# B&R Automation Studio project Splicer_V12_ACP10 (part 2)

#### slaveCyclic.st - Cyclic code
```iecst
(********************************************************************
 * COPYRIGHT -- Bernecker + Rainer
 ********************************************************************
 * Program: Slave_00
 * File: slaveCyclic.st
 * Author: Bernecker + Rainer
 * Created: March 01, 2011
 ********************************************************************
 * Implementation of program Slave_00
 ********************************************************************)

PROGRAM _CYCLIC

(************CHECK IF POWER SHOULD BE OFF ***************************)
    IF ((GlobalCommand.Power = FALSE) AND (Slave[SLAVE_INDEX].Command.Power = FALSE)) THEN
        SlaveStep := STATE_WAIT;
    END_IF

    (* central monitoring of the stop command allows a shorter reaction time *)
    IF ((GlobalCommand.Stop = TRUE) OR (Slave[SLAVE_INDEX].Command.Stop = TRUE)) THEN
        IF ((GlobalCommand.Power = TRUE) OR (Slave[SLAVE_INDEX].Command.Power = TRUE)) THEN
            SlaveStep := STATE_STOP;
            (* reset all FB execute inputs we use *)
            MC_Home_0.Execute := FALSE;
            MC_Halt_0.Execute := FALSE;
            MC_MoveAbsolute_0.Execute := FALSE;
            MC_MoveAdditive_0.Execute := FALSE;
            MC_MoveVelocity_0.Execute := FALSE;

            MC_BR_InitAutData_0.Execute := FALSE;
            MC_BR_AutCommand_0.Enable := FALSE;
            MC_BR_AutCommand_0.Start := FALSE;
            MC_BR_AutCommand_0.Restart := FALSE;
            MC_BR_AutCommand_0.Stop := FALSE;
            MC_BR_AutCommand_0.EndAutomat := FALSE;

            Slave[SLAVE_INDEX].Command.MoveJogPos := FALSE;
            Slave[SLAVE_INDEX].Command.MoveJogNeg := FALSE;
        END_IF
    END_IF

(************************** MC_READSTATUS ***************************)
MC_ReadStatus_0.Enable := NOT(MC_ReadStatus_0.Error);
MC_ReadStatus_0.Axis := SlaveRef[SLAVE_INDEX];
MC_ReadStatus_0();
Slave[SLAVE_INDEX].AxisState.Disabled             := MC_ReadStatus_0.Disabled;
Slave[SLAVE_INDEX].AxisState.StandStill           := MC_ReadStatus_0.StandStill;
Slave[SLAVE_INDEX].AxisState.Stopping             := MC_ReadStatus_0.Stopping;
Slave[SLAVE_INDEX].AxisState.Homing               := MC_ReadStatus_0.Homing;
Slave[SLAVE_INDEX].AxisState.DiscreteMotion       := MC_ReadStatus_0.DiscreteMotion;
Slave[SLAVE_INDEX].AxisState.ContinuousMotion     := MC_ReadStatus_0.ContinuousMotion;
Slave[SLAVE_INDEX].AxisState.SynchronizedMotion   := MC_ReadStatus_0.SynchronizedMotion;
Slave[SLAVE_INDEX].AxisState.ErrorStop            := MC_ReadStatus_0.Errorstop;

(********************** MC_BR_READDRIVESTATUS ***********************)
MC_BR_ReadDriveStatus_0.Enable := NOT(MC_BR_ReadDriveStatus_0.Error);
MC_BR_ReadDriveStatus_0.Axis := SlaveRef[SLAVE_INDEX];
MC_BR_ReadDriveStatus_0.AdrDriveStatus := ADR(Slave[SLAVE_INDEX].Status.DriveStatus);
MC_BR_ReadDriveStatus_0();

(********************* MC_READACTUALPOSITION ************************)
MC_ReadActualPosition_0.Enable := NOT(MC_ReadActualPosition_0.Error);
MC_ReadActualPosition_0.Axis := SlaveRef[SLAVE_INDEX];
MC_ReadActualPosition_0();
IF(MC_ReadActualPosition_0.Valid = TRUE) THEN
    Slave[SLAVE_INDEX].Status.ActPosition := MC_ReadActualPosition_0.Position;
END_IF

(********************* MC_READACTUALVELOCITY ************************)
MC_ReadActualVelocity_0.Enable := NOT(MC_ReadActualVelocity_0.Error);
MC_ReadActualVelocity_0.Axis := SlaveRef[SLAVE_INDEX];
MC_ReadActualVelocity_0();
IF(MC_ReadActualVelocity_0.Valid = TRUE) THEN
    Slave[SLAVE_INDEX].Status.ActVelocity := MC_ReadActualVelocity_0.Velocity;
END_IF

CASE SlaveStep OF
(****************************** WAIT ********************************)
    STATE_WAIT: (* STATE: Wait *)
        IF ((GlobalCommand.Power = TRUE) OR (Slave[SLAVE_INDEX].Command.Power = TRUE)) THEN
            SlaveStep := STATE_POWER_ON;
        ELSE
            MC_Power_0.Enable := FALSE;
        END_IF

        (* reset all FB execute inputs we use *)
        MC_Home_0.Execute := FALSE;
        MC_Halt_0.Execute := FALSE;
        MC_Stop_0.Execute := FALSE;
        MC_MoveAbsolute_0.Execute := FALSE;
        MC_MoveAdditive_0.Execute := FALSE;
        MC_MoveVelocity_0.Execute := FALSE;

        (* reset user commands *)
        Slave[SLAVE_INDEX].Command.Stop := FALSE;
        Slave[SLAVE_INDEX].Command.MoveJogPos := FALSE;
        Slave[SLAVE_INDEX].Command.MoveJogNeg := FALSE;
        Slave[SLAVE_INDEX].Command.MoveVelocity := FALSE;
        Slave[SLAVE_INDEX].Command.MoveAbsolute := FALSE;
        Slave[SLAVE_INDEX].Command.MoveAdditive := FALSE;

    (* End of STATE_WAIT *)

(****************************** POWER ON ****************************)
    STATE_POWER_ON: (* STATE: Power on *)
        IF (PowerSupplyOn = TRUE) THEN
            MC_Power_0.Enable := TRUE;
        END_IF
        IF (MC_Power_0.Status = TRUE) THEN
            SlaveStep := STATE_READY;
        END_IF

        (* if a power error occured switch off controller *)
        IF (MC_Power_0.Error = TRUE) THEN
            MC_Power_0.Enable := FALSE;
        END_IF

        (* End of STATE_POWER_ON *)

(****************************** READY *******************************)
    STATE_READY: (* STATE: Waiting for Commands *)
        IF ((Slave[SLAVE_INDEX].Command.Home = TRUE) OR (GlobalCommand.Home = TRUE)) THEN
            Slave[SLAVE_INDEX].Command.Home := FALSE;
            SlaveStep := STATE_HOME;
        ELSIF ((Slave[SLAVE_INDEX].Command.Stop = TRUE) OR (GlobalCommand.Stop = TRUE)) THEN
            SlaveStep := STATE_STOP;
        ELSIF (Slave[SLAVE_INDEX].Command.MoveJogPos = TRUE) THEN
            SlaveStep := STATE_JOG_POSITIVE;
        ELSIF (Slave[SLAVE_INDEX].Command.MoveJogNeg = TRUE) THEN
            SlaveStep := STATE_JOG_NEGATIVE;
        ELSIF (Slave[SLAVE_INDEX].Command.MoveAbsolute = TRUE) THEN
            Slave[SLAVE_INDEX].Command.MoveAbsolute := FALSE;
            SlaveStep := STATE_MOVE_ABSOLUTE;
        ELSIF (Slave[SLAVE_INDEX].Command.MoveAdditive = TRUE) THEN
            Slave[SLAVE_INDEX].Command.MoveAdditive := FALSE;
            SlaveStep := STATE_MOVE_ADDITIVE;
        ELSIF (Slave[SLAVE_INDEX].Command.MoveVelocity = TRUE) THEN
            Slave[SLAVE_INDEX].Command.MoveVelocity := FALSE;
            SlaveStep := STATE_MOVE_VELOCITY;
        ELSIF (Slave[SLAVE_INDEX].Command.Halt = TRUE) THEN
            Slave[SLAVE_INDEX].Command.Halt := FALSE;
            SlaveStep := STATE_HALT;
        ELSIF (Slave[SLAVE_INDEX].Command.StartAutomat = TRUE) THEN
            Slave[SLAVE_INDEX].Command.StartAutomat := FALSE;
            SlaveStep := STATE_AUTOMAT_INIT;
        ELSIF (Slave[SLAVE_INDEX].Command.RestartAutomat = TRUE) THEN
            Slave[SLAVE_INDEX].Command.RestartAutomat := FALSE;
            SlaveStep := STATE_AUTOMAT_RESTART;
        ELSIF (Slave[SLAVE_INDEX].Command.EndAutomat = TRUE) THEN
            Slave[SLAVE_INDEX].Command.EndAutomat := FALSE;
            SlaveStep := STATE_AUTOMAT_END;
        ELSIF (Slave[SLAVE_INDEX].Command.StopSlave = TRUE) THEN
            Slave[SLAVE_INDEX].Command.StopSlave := FALSE;
            SlaveStep := STATE_AUTOMAT_STOP;
        END_IF

        (* End of STATE_READY *)

(****************************** HOME ********************************)
    STATE_HOME: (* STATE: start homing process *)
        MC_Home_0.Position := Slave[SLAVE_INDEX].Parameter.HomePosition;
        MC_Home_0.HomingMode := Slave[SLAVE_INDEX].Parameter.HomeMode;
        MC_Home_0.Execute := TRUE;
        IF (MC_Home_0.Done = TRUE) THEN
            GlobalCommand.Home := FALSE;
            MC_Home_0.Execute := FALSE;
            SlaveStep := STATE_READY;
        END_IF

        (* if a homing error occured go to ready state *)
        IF ((MC_Home_0.Error = TRUE) OR (MC_Home_0.CommandAborted = TRUE)) THEN
            MC_Home_0.Execute := FALSE;
            SlaveStep := STATE_READY;
        END_IF

        (* End of STATE_HOME *)

(*************************** HALT MOVEMENT **************************)
    STATE_HALT: (* STATE: Stop the active movement *)
        MC_Halt_0.Deceleration := Slave[SLAVE_INDEX].Parameter.Deceleration;
        MC_Halt_0.Execute := TRUE;
        IF (MC_Halt_0.Done = TRUE) THEN
            MC_Halt_0.Execute := FALSE;
            SlaveStep := STATE_READY;
       END_IF

       (* check if error occured *)
       IF ((MC_Halt_0.Error = TRUE) OR (MC_Halt_0.CommandAborted = TRUE)) THEN
           MC_Halt_0.Execute := FALSE;
           SlaveStep := STATE_READY;
       END_IF

       (* End of STATE_HALT *)

(*************************** STOP MOVEMENT **************************)
    STATE_STOP: (* STATE: Stop movement as long as command is set *)
        MC_Stop_0.Deceleration := Slave[SLAVE_INDEX].Parameter.Deceleration;
        MC_Stop_0.Execute := TRUE;

        (* if axis is stopped go to ready state *)
        IF ((MC_Stop_0.Done = TRUE) AND (Slave[SLAVE_INDEX].Command.Stop = FALSE) AND (GlobalCommand.Stop = FALSE)) THEN
            MC_Stop_0.Execute := FALSE;
            SlaveStep := STATE_READY;
        END_IF

        (* check if error occured *)
        IF (((MC_Stop_0.Error = TRUE) OR (MC_Stop_0.CommandAborted = TRUE)) AND
             (Slave[SLAVE_INDEX].Command.Stop = FALSE) AND
             (GlobalCommand.Stop = FALSE)) THEN
            MC_Stop_0.Execute := FALSE;
            SlaveStep := STATE_READY;
        END_IF

       (* End of STATE_STOP *)

(******************* START JOG MOVEMENT POSITIVE ********************)
    STATE_JOG_POSITIVE: (* STATE: Start jog movement in positive direction *)
        MC_MoveVelocity_0.Velocity      := Slave[SLAVE_INDEX].Parameter.JogVelocity;
        MC_MoveVelocity_0.Acceleration  := Slave[SLAVE_INDEX].Parameter.Acceleration;
        MC_MoveVelocity_0.Deceleration  := Slave[SLAVE_INDEX].Parameter.Deceleration;
        MC_MoveVelocity_0.Direction     := mcPOSITIVE_DIR;
        MC_MoveVelocity_0.Execute := 1;

        (* check if jog movement should be stopped *)
        IF (Slave[SLAVE_INDEX].Command.MoveJogPos = FALSE) THEN
            MC_MoveVelocity_0.Execute := FALSE;
            SlaveStep := STATE_HALT;
        END_IF

        IF ((MC_MoveVelocity_0.Error = TRUE) OR (MC_MoveVelocity_0.CommandAborted = TRUE)) THEN
            MC_MoveVelocity_0.Execute := FALSE;
            SlaveStep := STATE_READY;
        END_IF

        (* End of STATE_JOG_POSITIVE *)

(********************START JOG MOVEMENT NEGATIVE ********************)
    STATE_JOG_NEGATIVE: (* STATE: Start jog movement in negative direction *)
        MC_MoveVelocity_0.Velocity      := Slave[SLAVE_INDEX].Parameter.JogVelocity;
        MC_MoveVelocity_0.Acceleration  := Slave[SLAVE_INDEX].Parameter.Acceleration;
        MC_MoveVelocity_0.Deceleration  := Slave[SLAVE_INDEX].Parameter.Deceleration;
        MC_MoveVelocity_0.Direction     := mcNEGATIVE_DIR;
        MC_MoveVelocity_0.Execute := 1;

        (* check if jog movement should be stopped *)
        IF (Slave[SLAVE_INDEX].Command.MoveJogNeg = FALSE) THEN
            MC_MoveVelocity_0.Execute := FALSE;
            SlaveStep := STATE_HALT;
        END_IF

        IF ((MC_MoveVelocity_0.Error = TRUE) OR (MC_MoveVelocity_0.CommandAborted = TRUE)) THEN
            MC_MoveVelocity_0.Execute := FALSE;
            SlaveStep := STATE_READY;
        END_IF

        (* End of STATE_JOG_NEGATIVE *)

(********************* START ABSOLUTE MOVEMENT **********************)
    STATE_MOVE_ABSOLUTE: (* STATE: Start absolute movement *)
        MC_MoveAbsolute_0.Position      := Slave[SLAVE_INDEX].Parameter.Position;
        MC_MoveAbsolute_0.Velocity      := Slave[SLAVE_INDEX].Parameter.Velocity;
        MC_MoveAbsolute_0.Acceleration  := Slave[SLAVE_INDEX].Parameter.Acceleration;
        MC_MoveAbsolute_0.Deceleration  := Slave[SLAVE_INDEX].Parameter.Deceleration;
        MC_MoveAbsolute_0.Direction     := Slave[SLAVE_INDEX].Parameter.Direction;
        MC_MoveAbsolute_0.Execute := 1;

        IF (Slave[SLAVE_INDEX].Command.Halt = TRUE) THEN
            Slave[SLAVE_INDEX].Command.Halt := 0;
            MC_MoveAbsolute_0.Execute := 0;
            SlaveStep := STATE_HALT;
        ELSIF (MC_MoveAbsolute_0.Done = TRUE) THEN
            MC_MoveAbsolute_0.Execute := FALSE;
            SlaveStep := STATE_READY;
        END_IF

        IF ((MC_MoveAbsolute_0.Error = TRUE) OR (MC_MoveAbsolute_0.CommandAborted = TRUE)) THEN
            MC_MoveAbsolute_0.Execute := FALSE;
            SlaveStep := STATE_READY;
        END_IF

        (* End of STATE_MOVE_ABSOLUTE *)

(********************* START ADDITIVE MOVEMENT **********************)
    STATE_MOVE_ADDITIVE: (* STATE: Start additive movement *)
        MC_MoveAdditive_0.Distance      := Slave[SLAVE_INDEX].Parameter.Distance;
        MC_MoveAdditive_0.Velocity      := Slave[SLAVE_INDEX].Parameter.Velocity;
        MC_MoveAdditive_0.Acceleration  := Slave[SLAVE_INDEX].Parameter.Acceleration;
        MC_MoveAdditive_0.Deceleration  := Slave[SLAVE_INDEX].Parameter.Deceleration;
        MC_MoveAdditive_0.Execute := 1;
        IF (Slave[SLAVE_INDEX].Command.Halt = TRUE) THEN
            Slave[SLAVE_INDEX].Command.Halt := FALSE;
            MC_MoveAdditive_0.Execute := FALSE;
            SlaveStep := STATE_HALT;
        ELSIF (MC_MoveAdditive_0.Done = TRUE) THEN
            MC_MoveAdditive_0.Execute := FALSE;
             SlaveStep := STATE_READY;
        END_IF

        (* check IF error occured *)
        IF ((MC_MoveAdditive_0.Error = TRUE) OR (MC_MoveAdditive_0.CommandAborted = TRUE)) THEN
            MC_MoveAdditive_0.Execute := FALSE;
            SlaveStep := STATE_READY;
        END_IF

        (* End of STATE_MOVE_ADDITIVE *)

(********************* START VELOCITY MOVEMENT **********************)
    STATE_MOVE_VELOCITY: (* STATE: Start velocity movement *)
        MC_MoveVelocity_0.Velocity      := Slave[SLAVE_INDEX].Parameter.Velocity;
        MC_MoveVelocity_0.Acceleration  := Slave[SLAVE_INDEX].Parameter.Acceleration;
        MC_MoveVelocity_0.Deceleration  := Slave[SLAVE_INDEX].Parameter.Deceleration;
        MC_MoveVelocity_0.Direction     := Slave[SLAVE_INDEX].Parameter.Direction;
        MC_MoveVelocity_0.Execute := 1;

        IF (Slave[SLAVE_INDEX].Command.Halt = TRUE) THEN
            Slave[SLAVE_INDEX].Command.Halt := FALSE;
            MC_MoveVelocity_0.Execute := FALSE;
            SlaveStep := STATE_HALT;
        ELSIF (MC_MoveVelocity_0.InVelocity = TRUE) THEN
            MC_MoveVelocity_0.Execute := FALSE;
             SlaveStep := STATE_READY;
        END_IF
        (* check if error occured *)
        IF ((MC_MoveVelocity_0.Error = TRUE) OR (MC_MoveVelocity_0.CommandAborted = TRUE)) THEN
            MC_MoveVelocity_0.Execute := FALSE;
            SlaveStep := STATE_READY;
        END_IF

        (* End of STATE_MOVE_ADDITIVE *)

(****************** INITIALIZE AUTOMAT PARAMETERS *******************)
    STATE_AUTOMAT_INIT:
        Labeler(MasterRef[0],AutData); (*Call of the function with the Automat Data*)

        MC_BR_InitAutData_0.InitOptions.GlobalParams      := mcALL_PARAMS;
        MC_BR_InitAutData_0.InitOptions.StateIndex        := mcALL_STATES;
        MC_BR_InitAutData_0.InitOptions.EventIndex        := mcALL_EVENTS;
        MC_BR_InitAutData_0.InitOptions.MaxStatesPerCycle := 14;
        MC_BR_InitAutData_0.InitOptions.Force             := mcOFF;
        MC_BR_InitAutData_0.AdrAutData  := ADR(AutData);
        MC_BR_InitAutData_0.Execute     := TRUE;

        (* wait for initialization done *)
        IF (MC_BR_InitAutData_0.Done = TRUE) THEN
            MC_BR_InitAutData_0.Execute := FALSE;
            SlaveStep := STATE_AUTOMAT_START;
        END_IF

        (* check if error occured *)
        IF (MC_BR_InitAutData_0.Error = TRUE) THEN
            MC_BR_InitAutData_0.Execute := FALSE;
            SlaveStep := STATE_READY;
        END_IF

        (* End of STATE_MOVE_VELOCITY *)

(********************** ENABLE CAM-AUTOMAT **************************)
    STATE_AUTOMAT_START:
        MC_BR_AutCommand_0.Enable := TRUE;
        MC_BR_AutCommand_0.Start := TRUE;

        (* wait for autoamt stop *)
        IF (Slave[SLAVE_INDEX].Command.Halt = TRUE) THEN
            Slave[SLAVE_INDEX].Command.Halt := FALSE;
            MC_BR_AutCommand_0.Enable := FALSE;
            MC_BR_AutCommand_0.Start := FALSE;
            SlaveStep := STATE_HALT;
        ELSIF (MC_BR_AutCommand_0.Running = TRUE) THEN
            MC_BR_AutCommand_0.Start := FALSE;
            SlaveStep := STATE_READY;
        END_IF

        (* check if error occured *)
        IF (MC_BR_AutCommand_0.Error = TRUE) THEN
            MC_BR_AutCommand_0.Enable := FALSE;
            MC_BR_AutCommand_0.Start := FALSE;
            SlaveStep := STATE_READY;
        END_IF

        (* End of STATE_AUTOMAT_START *)

(********************** RESTART CAM-AUTOMAT *************************)
    STATE_AUTOMAT_RESTART:
        IF (MC_BR_AutCommand_0.StandBy = FALSE) THEN
            SlaveStep := STATE_READY;
            RETURN;
        END_IF

        MC_BR_AutCommand_0.Enable := TRUE;
        MC_BR_AutCommand_0.Restart := TRUE;

        (* wait for autoamt stop *)
        IF (Slave[SLAVE_INDEX].Command.Halt = TRUE) THEN
            Slave[SLAVE_INDEX].Command.Halt := FALSE;
            MC_BR_AutCommand_0.Enable := FALSE;
            MC_BR_AutCommand_0.Restart := FALSE;
            SlaveStep := STATE_HALT;
        ELSIF (MC_BR_AutCommand_0.Running = TRUE) THEN
            MC_BR_AutCommand_0.Restart := FALSE;
            SlaveStep := STATE_READY;
        END_IF

        (* check if error occured *)
        IF (MC_BR_AutCommand_0.Error = TRUE) THEN
            MC_BR_AutCommand_0.Enable := FALSE;
            MC_BR_AutCommand_0.Restart := FALSE;
            SlaveStep := STATE_READY;
        END_IF

        (* End of STATE_AUTOMAT_RESTART *)

(*********************** STOP CAM-AUTOMAT ***************************)
    STATE_AUTOMAT_STOP:
        MC_BR_AutCommand_0.Deceleration := Slave[SLAVE_INDEX].Parameter.Deceleration;
        MC_BR_AutCommand_0.Stop := TRUE;

        (* check if automat is stopped *)
        IF (MC_BR_AutCommand_0.Running = FALSE) THEN
            MC_BR_AutCommand_0.Stop := FALSE;
            SlaveStep := STATE_READY;
        END_IF

        IF (MC_BR_AutCommand_0.Error = TRUE) THEN
            MC_BR_AutCommand_0.Enable := FALSE;
            MC_BR_AutCommand_0.Stop := FALSE;
            SlaveStep := STATE_READY;
        END_IF

        (* End of STATE_AUTOMAT_STOP *)

(************************ END CAM-AUTOMAT ***************************)
    STATE_AUTOMAT_END:
        MC_BR_AutCommand_0.Deceleration := Slave[SLAVE_INDEX].Parameter.Deceleration;
        MC_BR_AutCommand_0.Stop := TRUE;

        (* check if automat is stopped *)
        IF (MC_BR_AutCommand_0.Running = FALSE) THEN
            MC_BR_AutCommand_0.Enable := FALSE;
            MC_BR_AutCommand_0.EndAutomat := FALSE;
            SlaveStep := STATE_READY;
        END_IF

        (* check if error occured *)
        IF (MC_BR_AutCommand_0.Error = TRUE) THEN
            MC_BR_AutCommand_0.Enable := FALSE;
            MC_BR_AutCommand_0.EndAutomat := FALSE;
            SlaveStep := STATE_READY;
        END_IF

        (* End of STATE_AUTOMAT_STOP *)

(*********************** SEQUENCE END *******************************)
END_CASE

(*********************************************************************
        Function Block Calls
*********************************************************************)

(*************************** MC_POWER *******************************)
MC_Power_0.Axis := SlaveRef[SLAVE_INDEX];
MC_Power_0();

(**************************** MC_HOME *******************************)
MC_Home_0.Axis := SlaveRef[SLAVE_INDEX];
MC_Home_0();

(************************ MC_MOVEABSOLUTE ***************************)
MC_MoveAbsolute_0.Axis := SlaveRef[SLAVE_INDEX];
MC_MoveAbsolute_0();

(************************ MC_MOVEADDITIVE ***************************)
MC_MoveAdditive_0.Axis := SlaveRef[SLAVE_INDEX];
MC_MoveAdditive_0();

(************************ MC_MOVEVELOCITY ***************************)
MC_MoveVelocity_0.Axis := SlaveRef[SLAVE_INDEX];
MC_MoveVelocity_0();

(**************************** MC_STOP *******************************)
MC_Stop_0.Axis := SlaveRef[SLAVE_INDEX];
MC_Stop_0();

(*************************** MC_HALT ********************************)
MC_Halt_0.Axis := SlaveRef[SLAVE_INDEX];
MC_Halt_0();

(********************** MC_BR_INITAUTDATA ***************************)
MC_BR_InitAutData_0.Slave := SlaveRef[SLAVE_INDEX];
MC_BR_InitAutData_0();

(*********************** MC_BR_AUTCOMMAND ***************************)
MC_BR_AutCommand_0.SetSignal1 := Slave[SLAVE_INDEX].Command.SetSignal1;
MC_BR_AutCommand_0.SetSignal2 := Slave[SLAVE_INDEX].Command.SetSignal2;
MC_BR_AutCommand_0.SetSignal3 := Slave[SLAVE_INDEX].Command.SetSignal3;
MC_BR_AutCommand_0.SetSignal4 := Slave[SLAVE_INDEX].Command.SetSignal4;
MC_BR_AutCommand_0.ResetSignal1 := Slave[SLAVE_INDEX].Command.ResetSignal1;
MC_BR_AutCommand_0.ResetSignal2 := Slave[SLAVE_INDEX].Command.ResetSignal2;
MC_BR_AutCommand_0.ResetSignal3 := Slave[SLAVE_INDEX].Command.ResetSignal3;
MC_BR_AutCommand_0.ResetSignal4 := Slave[SLAVE_INDEX].Command.ResetSignal4;
MC_BR_AutCommand_0.Slave := SlaveRef[SLAVE_INDEX];
MC_BR_AutCommand_0();
Slave[SLAVE_INDEX].Status.AutomatRunning := MC_BR_AutCommand_0.Running;
Slave[SLAVE_INDEX].Status.AutomatStandBy := MC_BR_AutCommand_0.StandBy;
Slave[SLAVE_INDEX].Status.ActualStateIndex := MC_BR_AutCommand_0.ActualStateIndex;
Slave[SLAVE_INDEX].Status.ActualStateCamIndex := MC_BR_AutCommand_0.ActualStateCamIndex;
Slave[SLAVE_INDEX].Status.InCam := MC_BR_AutCommand_0.InCam;
Slave[SLAVE_INDEX].Status.InCompensation := MC_BR_AutCommand_0.InCompensation;
END_PROGRAM
```

#### slaveInit.st - Initialization code
```iecst
(********************************************************************
 * COPYRIGHT -- Bernecker + Rainer
 ********************************************************************
 * Program: Slave_00
 * File: slaveInit.st
 * Author: Bernecker + Rainer
 * Created: March 01, 2011
 ********************************************************************
 * Implementation of program Slave_00
 ********************************************************************)

PROGRAM _INIT
SlaveStep := STATE_WAIT; (* start step *)

Slave[SLAVE_INDEX].Parameter.Velocity       := 1000; (* velocity for movement *)
Slave[SLAVE_INDEX].Parameter.Acceleration   := 5000; (* acceleration for movement *)
Slave[SLAVE_INDEX].Parameter.Deceleration   := 5000; (* deceleration for movement *)
Slave[SLAVE_INDEX].Parameter.JogVelocity    := 400;  (* velocity for jogging *)
END_PROGRAM
```

#### slave.var - Local variables
```iecst
(*Actual step inside step sequencer*)
VAR
	SlaveStep : USINT; (*current  step in the step sequence*)
END_VAR
VAR CONSTANT
	STATE_WAIT : USINT := 0; (*constant for a waiting step*)
	STATE_POWER_ON : USINT := 1; (*constant for the step in which the controller is switched on*)
	STATE_HOME : USINT := 2; (*constant for the step in which the axis is referenced*)
	STATE_READY : USINT := 10; (*constant for a waiting step*)
	STATE_HALT : USINT := 11; (*constant for the step in which movements are stopped*)
	STATE_STOP : USINT := 12; (*constant for the step in which movements are stopped*)
	STATE_JOG_POSITIVE : USINT := 13; (*constant for the step in which positive jogging movement is executed*)
	STATE_JOG_NEGATIVE : USINT := 14; (*constant for the step in which negative jogging movement is executed*)
	STATE_MOVE_ABSOLUTE : USINT := 15; (*constant for the step in which a movement to defined position is executed*)
	STATE_MOVE_ADDITIVE : USINT := 16; (*constant for the step in which a movement with defined distance is executed*)
	STATE_MOVE_VELOCITY : USINT := 17; (*constant for the step in which a movement with defined velocity is started*)
	STATE_AUTOMAT_INIT : USINT := 30; (*constant for the step in which the automat is configured*)
	STATE_AUTOMAT_START : USINT := 31; (*constant for the step in which the automat is started*)
	STATE_AUTOMAT_STOP : USINT := 32; (*constant for the step in which the automat is stopped*)
	STATE_AUTOMAT_RESTART : USINT := 33; (*constant for the step in which the automat is restarted*)
	STATE_AUTOMAT_END : USINT := 34; (*constant for the step in which the automat is finished*)
END_VAR
(*Index of the used axis*)
VAR CONSTANT
	SLAVE_INDEX : USINT := 0; (*Index of the used axis*)
END_VAR
(*Configuration data of the automat*)
VAR
	AutData : MC_AUTDATA_TYP; (*configuration of the automat*)
END_VAR
(*Function Blocks*)
VAR
	MC_BR_AutCommand_0 : MC_BR_AutCommand; (*Function Block*)
	MC_BR_InitAutData_0 : MC_BR_InitAutData; (*Function Block*)
	MC_BR_ReadDriveStatus_0 : MC_BR_ReadDriveStatus; (*Function Block *)
	MC_Halt_0 : MC_Halt; (*Function Block *)
	MC_Home_0 : MC_Home; (*Function Block *)
	MC_MoveAbsolute_0 : MC_MoveAbsolute; (*Function Block *)
	MC_MoveAdditive_0 : MC_MoveAdditive; (*Function Block *)
	MC_MoveVelocity_0 : MC_MoveVelocity; (*Function Block *)
	MC_Power_0 : MC_Power; (*Function Block *)
	MC_ReadActualPosition_0 : MC_ReadActualPosition; (*Function Block *)
	MC_ReadActualVelocity_0 : MC_ReadActualVelocity; (*Function Block *)
	MC_ReadStatus_0 : MC_ReadStatus; (*Function Block *)
	MC_Stop_0 : MC_Stop; (*Function Block *)
END_VAR
```

#### slave.fun - functions
```iecst
(********************************************************************
 * COPYRIGHT -- Bernecker + Rainer
 ********************************************************************
 * Program: Slave_00
 * File: Slave_00.fun
 * Author: reischlj
 * Created: March 09, 2011
 ********************************************************************
 * Functions and function blocks of program Slave_00
 ********************************************************************)

FUNCTION Labeler : BOOL
	VAR_INPUT
		Axis : UDINT;
	END_VAR
	VAR_IN_OUT
		AutData : MC_AUTDATA_TYP;
	END_VAR
END_FUNCTION

FUNCTION CrossCutter : BOOL
	VAR_INPUT
		Axis : UDINT;
	END_VAR
	VAR_IN_OUT
		AutData : MC_AUTDATA_TYP;
	END_VAR
END_FUNCTION

FUNCTION FlyingSaw : BOOL
	VAR_INPUT
		Axis  : UDINT;
	END_VAR
	VAR_IN_OUT
		AutData : MC_AUTDATA_TYP;
	END_VAR
END_FUNCTION
```

#### Labeler.st - function
```iecst
(********************************************************************
 * COPYRIGHT -- Bernecker + Rainer
 ********************************************************************
 * PROGRAM: Slave
 * File: Labeler.st
 * Author: Bernecker + Rainer
 * Created: March 01, 2011
 *******************************************************************)

FUNCTION Labeler
    (*general automat parameter*)
        AutData.Master              := Axis;

        AutData.MaxMasterVelocity   := 1000;

    (*Automat STATE 0 Basis State*)

        AutData.State[0].Event[0].Type      := ncST_END;

        AutData.State[0].Event[0].Attribute := ncAT_ONCE;

        AutData.State[0].Event[0].NextState := 1;

    (*Automat STATE 1 Standstill*)

        AutData.State[1].CamProfileIndex    := 16#FFFF;

        AutData.State[1].MasterFactor       := 200;

        AutData.State[1].SlaveFactor        := 0;

        AutData.State[1].CompMode           := ncONLYCOMP;

        AutData.State[1].MasterCompDistance := 800;

        AutData.State[1].SlaveCompDistance  := 0;

        AutData.State[1].Event[0].Type      := ncTRIGGER1+ncP_EDGE;

        AutData.State[1].Event[0].Attribute := ncST_END;

        AutData.State[1].Event[0].NextState := 2;

        AutData.State[1].Event[1].Type      := ncST_END;

        AutData.State[1].Event[1].Attribute := ncST_END;

        AutData.State[1].Event[1].NextState := 1;

    (*Automat STATE 2 Labeling with half compensation*)

        AutData.State[2].CamProfileIndex    := 16#FFFF;

        AutData.State[2].MasterFactor       := 200;

        AutData.State[2].SlaveFactor        := 200;

        AutData.State[2].CompMode           := ncONLYCOMP;
        AutData.State[2].MasterCompDistance := 800;

        AutData.State[2].SlaveCompDistance  := 400;

        AutData.State[2].Event[0].Type      := ncTRIGGER1+ncP_EDGE;

        AutData.State[2].Event[0].Attribute := ncST_END;

        AutData.State[2].Event[0].NextState := 3;

        AutData.State[2].Event[1].Type      := ncST_END;

        AutData.State[2].Event[1].Attribute := ncST_END;

        AutData.State[2].Event[1].NextState := 4;

    (*Automat STATE 3 Labeling *)

        AutData.State[3].CamProfileIndex    := 16#FFFF;

        AutData.State[3].MasterFactor       := 200;

        AutData.State[3].SlaveFactor        := 200;

        AutData.State[3].CompMode           := ncONLYCOMP;

        AutData.State[3].MasterCompDistance := 800;

        AutData.State[3].SlaveCompDistance  := 800;

        AutData.State[3].Event[0].Type      := ncTRIGGER1+ncP_EDGE;

        AutData.State[3].Event[0].Attribute := ncST_END;

        AutData.State[3].Event[0].NextState := 3;

        AutData.State[3].Event[1].Type      := ncST_END;
		AutData.State[3].Event[1].Attribute := ncST_END;
		AutData.State[3].Event[1].NextState := 4;

    (*Automat STATE 4 Return to starting position*)
        AutData.State[4].CamProfileIndex    := 16#FFFF;
        AutData.State[4].MasterFactor       := 200;
        AutData.State[4].SlaveFactor        := 0;
        AutData.State[4].CompMode           := ncONLYCOMP;
        AutData.State[4].MasterCompDistance := 800;
        AutData.State[4].SlaveCompDistance  := 400;

        AutData.State[4].Event[0].Type      := ncTRIGGER1+ncP_EDGE;
        AutData.State[4].Event[0].Attribute := ncST_END;
        AutData.State[4].Event[0].NextState := 2;

        AutData.State[4].Event[1].Type      := ncST_END;
        AutData.State[4].Event[1].Attribute := ncST_END;
        AutData.State[4].Event[1].NextState := 1;

        Labeler := TRUE;
END_FUNCTION
```

#### CrossCutter.st - function
```iecst
(********************************************************************
 * COPYRIGHT -- Bernecker + Rainer
 ********************************************************************
 * PROGRAM: Slave
 * File: CrossCutter.st
 * Author: Bernecker + Rainer
 * Created: March 01, 2011
 *******************************************************************)

FUNCTION CrossCutter
    (*general automat parameter*)
        AutData.Master              := Axis;

        AutData.MaxMasterVelocity   := 1000;

    (*Automat STATE 0 Basis State*)

        AutData.State[0].Event[0].Type      := ncST_END;

        AutData.State[0].Event[0].Attribute := ncAT_ONCE;

        AutData.State[0].Event[0].NextState := 1;

    (*Automat STATE 1 Standstill*)

        AutData.State[1].CamProfileIndex    := 16#FFFE;

        AutData.State[1].MasterFactor       := 200;

        AutData.State[1].SlaveFactor        := 0;
        AutData.State[1].CompMode           := ncWITH_CAM;
        AutData.State[1].MasterCompDistance := 1000;
        AutData.State[1].SlaveCompDistance  := 0;

        AutData.State[1].Event[0].Type      := ncSIGNAL1;
        AutData.State[1].Event[0].Attribute := ncAT_ONCE;
        AutData.State[1].Event[0].NextState := 2;

    (*Automat STATE 2 Move Slave to Cutting Position*)
        AutData.State[2].CamProfileIndex    := 16#FFFF;
        AutData.State[2].MasterFactor       := 200;
        AutData.State[2].SlaveFactor        := 200;
        AutData.State[2].CompMode           := ncWITH_CAM;
        AutData.State[2].MasterCompDistance := 500;
        AutData.State[2].SlaveCompDistance  := 1800;

        AutData.State[2].Event[0].Type      := ncST_END;
        AutData.State[2].Event[0].Attribute := ncST_END;
        AutData.State[2].Event[0].NextState := 3;

    (*Automat STATE 3 Execute one cut every master period*)
        AutData.State[3].CamProfileIndex    := 16#FFFF;
        AutData.State[3].MasterFactor       := 200;
        AutData.State[3].SlaveFactor        := 200;
        AutData.State[3].CompMode           := ncWITH_CAM;
        AutData.State[3].MasterCompDistance := 1000;
        AutData.State[3].SlaveCompDistance  := 3600;

        AutData.State[3].Event[0].Type      := ncSIGNAL2;
        AutData.State[3].Event[0].Attribute := ncST_END;
        AutData.State[3].Event[0].NextState := 4;

        AutData.State[3].Event[1].Type      := ncST_END;
        AutData.State[3].Event[1].Attribute := ncST_END;
        AutData.State[3].Event[1].NextState := 3;

    (*Automat STATE 4 Stop Motion at Starting Point*)
        AutData.State[4].CamProfileIndex    := 16#FFFF;
        AutData.State[4].MasterFactor       := 200;
        AutData.State[4].SlaveFactor        := 0;
        AutData.State[4].CompMode           := ncWITH_CAM;
        AutData.State[4].MasterCompDistance := 500;
        AutData.State[4].SlaveCompDistance  := 1800;

        AutData.State[4].Event[0].Type      := ncST_END;
        AutData.State[4].Event[0].Attribute := ncST_END;
        AutData.State[4].Event[0].NextState := 1;

        CrossCutter := TRUE;
END_FUNCTION
```

#### FlyingSaw.st - function
```iecst
(********************************************************************
 * COPYRIGHT -- Bernecker + Rainer
 ********************************************************************
 * PROGRAM: Slave
 * File: FlyingSaw.st
 * Author: Bernecker + Rainer
 * Created: March 01, 2011
 *******************************************************************)

FUNCTION FlyingSaw
    (*general automat parameters*)
        AutData.Master              := Axis;

        AutData.StartPosition       := 0;

        AutData.StartInterval       := 1000;

        AutData.MaxMasterVelocity   := 1000;

    (*Automat STATE 0 Basis State*)

        AutData.State[0].Event[0].Type      := ncST_END;

        AutData.State[0].Event[0].Attribute := ncAT_ONCE;

        AutData.State[0].Event[0].NextState := 1;

    (*Automat STATE 1 Standstill*)

        AutData.State[1].CamProfileIndex    := 16#FFFF;

        AutData.State[1].MasterFactor       := 200;

        AutData.State[1].SlaveFactor        := 0;

        AutData.State[1].CompMode           := ncONLYCOMP;

        AutData.State[1].MasterCompDistance := 800;

        AutData.State[1].SlaveCompDistance  := 0;

        AutData.State[1].Event[0].Type      := ncS_START;

        AutData.State[1].Event[0].Attribute := ncAT_ONCE;

        AutData.State[1].Event[0].NextState := 2;

    (*Autoamt STATE 2 Synchronous movement*)
        AutData.State[2].CamProfileIndex    := 16#FFFF;
        AutData.State[2].MasterFactor       := 500;
        AutData.State[2].SlaveFactor        := 500;
        AutData.State[2].CompMode           := ncONLYCOMP;
        AutData.State[2].MasterCompDistance := 100;
        AutData.State[2].SlaveCompDistance  := 100;

        AutData.State[2].Event[0].Type      := ncST_END;
        AutData.State[2].Event[0].Attribute := ncST_END;
        AutData.State[2].Event[0].NextState := 3;

    (*Automat STATE 3 Return to starting position*)
        AutData.State[3].CamProfileIndex    := 16#FFFF;
        AutData.State[3].MasterFactor       := 100;
        AutData.State[3].SlaveFactor        := 0;
        AutData.State[3].CompMode           := ncONLYCOMP;
        AutData.State[3].MasterCompDistance := 800;
        AutData.State[3].SlaveCompDistance  := -600;

        AutData.State[3].Event[0].Type      := ncST_END;
        AutData.State[3].Event[0].Attribute := ncST_END;
        AutData.State[3].Event[0].NextState := 1;

        FlyingSaw := TRUE;
END_FUNCTION
```

### Program Logical/Template/Logical/LibACP10MC_MotionControl_ST/ErrorHandling (IEC) - error handling task

#### errorHandlingCyclic.st - Cyclic code
```iecst
(********************************************************************
 * COPYRIGHT -- Bernecker + Rainer
 ********************************************************************
 * Program: ErrorHandling
 * File: errorHandlingCyclic.st
 * Author: Bernecker + Rainer
 * Created: March 01, 2011
 ********************************************************************
 * Implementation of program Errorhandling
 ********************************************************************)

PROGRAM _CYCLIC

(******************************ERROR_CHECK***************************)
(* check if one of the used FBs reports an error *)
IF ((MC_BR_AxisErrorCollector_0.Error = TRUE) OR (MC_Reset_0.Error = TRUE)) THEN
    ErrorStep := STATE_INTERNAL_ERROR;
END_IF

FOR configAxisIndex := 0 TO TOTAL_AXES BY 1 DO
    IF ((MC_BR_ReadAxisError_0[configAxisIndex].Error = TRUE) OR (MC_ReadStatus_0[configAxisIndex].Error = TRUE)) THEN
        ErrorStep := STATE_INTERNAL_ERROR;
        EXIT;
    END_IF
END_FOR

CASE ErrorStep OF

(**************************** CONFIGURATE_FBS ***********************)
    STATE_CONFIG_FBS: (* configurate the used FBs for the error handling *)
        MC_BR_AxisErrorCollector_0.Axis := mcALL_AXES;
        MC_BR_AxisErrorCollector_0.Enable := TRUE;

        (* configuration the MC_BR_ReadAxisError_0-FBs for all single axes *)
        FOR axisIndex := 0 TO (AXIS_MAX_INDEX) BY 1 DO
            MC_BR_ReadAxisError_0[axisIndex].Axis := AxisRef[axisIndex];
            MC_BR_ReadAxisError_0[axisIndex].Enable := TRUE;
            MC_BR_ReadAxisError_0[axisIndex].Configuration.Format := mcWRAP;
            MC_BR_ReadAxisError_0[axisIndex].Configuration.LineLength := SIZEOF(Axis[axisIndex].Error.ErrorText[0]);
            MC_BR_ReadAxisError_0[axisIndex].Configuration.DataLength := SIZEOF(Axis[axisIndex].Error.ErrorText);
            MC_BR_ReadAxisError_0[axisIndex].Configuration.DataAddress := ADR(Axis[axisIndex].Error.ErrorText[0]);
            MC_BR_ReadAxisError_0[axisIndex].Configuration.DataObjectName :='acp10etxen';
            MC_BR_ReadAxisError_0[axisIndex].Mode := mcTEXT;

            MC_ReadStatus_0[axisIndex].Axis := AxisRef[axisIndex];
            MC_ReadStatus_0[axisIndex].Enable := TRUE;
        END_FOR

        (* configuration the MC_BR_ReadAxisError_0-FBs for all master axes *)
        FOR masterIndex := 0 TO (MASTER_MAX_INDEX) BY 1 DO
            MC_BR_ReadAxisError_0[masterIndex+AXIS_NUMBER].Axis := MasterRef[masterIndex];
            MC_BR_ReadAxisError_0[masterIndex+AXIS_NUMBER].Enable := TRUE;
            MC_BR_ReadAxisError_0[masterIndex+AXIS_NUMBER].Configuration.Format := mcWRAP;
            MC_BR_ReadAxisError_0[masterIndex+AXIS_NUMBER].Configuration.LineLength := SIZEOF(Master[masterIndex].Error.ErrorText[0]);
            MC_BR_ReadAxisError_0[masterIndex+AXIS_NUMBER].Configuration.DataLength := SIZEOF(Master[masterIndex].Error.ErrorText);
            MC_BR_ReadAxisError_0[masterIndex+AXIS_NUMBER].Configuration.DataAddress := ADR(Master[masterIndex].Error.ErrorText[0]);
            MC_BR_ReadAxisError_0[masterIndex+AXIS_NUMBER].Configuration.DataObjectName := 'acp10etxen';
            MC_BR_ReadAxisError_0[masterIndex+AXIS_NUMBER].Mode := mcTEXT;

            MC_ReadStatus_0[masterIndex+AXIS_NUMBER].Axis := MasterRef[masterIndex];
            MC_ReadStatus_0[masterIndex+AXIS_NUMBER].Enable := TRUE;
        END_FOR

        (* configuration the MC_BR_ReadAxisError_0-FBs for all slave axes *)
        FOR slaveIndex := 0 TO (SLAVE_MAX_INDEX) BY 1 DO
            MC_BR_ReadAxisError_0[slaveIndex+AXIS_NUMBER+MASTER_NUMBER].Axis := SlaveRef[slaveIndex];
            MC_BR_ReadAxisError_0[slaveIndex+AXIS_NUMBER+MASTER_NUMBER].Enable := TRUE;
            MC_BR_ReadAxisError_0[slaveIndex+AXIS_NUMBER+MASTER_NUMBER].Configuration.Format := mcWRAP;
            MC_BR_ReadAxisError_0[slaveIndex+AXIS_NUMBER+MASTER_NUMBER].Configuration.LineLength := SIZEOF(Slave[slaveIndex].Error.ErrorText[0]);
            MC_BR_ReadAxisError_0[slaveIndex+AXIS_NUMBER+MASTER_NUMBER].Configuration.DataLength := SIZEOF(Slave[slaveIndex].Error.ErrorText);
            MC_BR_ReadAxisError_0[slaveIndex+AXIS_NUMBER+MASTER_NUMBER].Configuration.DataAddress := ADR(Slave[slaveIndex].Error.ErrorText[0]);
            MC_BR_ReadAxisError_0[slaveIndex+AXIS_NUMBER+MASTER_NUMBER].Configuration.DataObjectName := 'acp10etxen';
            MC_BR_ReadAxisError_0[slaveIndex+AXIS_NUMBER+MASTER_NUMBER].Mode := mcTEXT;

            MC_ReadStatus_0[slaveIndex+AXIS_NUMBER+MASTER_NUMBER].Axis := SlaveRef[slaveIndex];
            MC_ReadStatus_0[slaveIndex+AXIS_NUMBER+MASTER_NUMBER].Enable := TRUE;
        END_FOR

        (* configuration the MC_BR_ReadAxisError_0-FBs for all power supply module *)
        FOR psmIndex := 0 TO (PSM_MAX_INDEX) BY 1 DO
            MC_BR_ReadAxisError_0[psmIndex+AXIS_NUMBER+MASTER_NUMBER+SLAVE_NUMBER].Axis := PsmRef[psmIndex];
            MC_BR_ReadAxisError_0[psmIndex+AXIS_NUMBER+MASTER_NUMBER+SLAVE_NUMBER].Enable := TRUE;
            MC_BR_ReadAxisError_0[psmIndex+AXIS_NUMBER+MASTER_NUMBER+SLAVE_NUMBER].Configuration.Format := mcWRAP;
            MC_BR_ReadAxisError_0[psmIndex+AXIS_NUMBER+MASTER_NUMBER+SLAVE_NUMBER].Configuration.LineLength := SIZEOF(PowerSupply[psmIndex].Error.ErrorText[0]);
            MC_BR_ReadAxisError_0[psmIndex+AXIS_NUMBER+MASTER_NUMBER+SLAVE_NUMBER].Configuration.DataLength := SIZEOF(PowerSupply[psmIndex].Error.ErrorText);
            MC_BR_ReadAxisError_0[psmIndex+AXIS_NUMBER+MASTER_NUMBER+SLAVE_NUMBER].Configuration.DataAddress := ADR(PowerSupply[psmIndex].Error.ErrorText[0]);
            MC_BR_ReadAxisError_0[psmIndex+AXIS_NUMBER+MASTER_NUMBER+SLAVE_NUMBER].Configuration.DataObjectName := 'acp10etxen';
            MC_BR_ReadAxisError_0[psmIndex+AXIS_NUMBER+MASTER_NUMBER+SLAVE_NUMBER].Mode := mcTEXT;

            MC_ReadStatus_0[psmIndex+AXIS_NUMBER+MASTER_NUMBER+SLAVE_NUMBER].Axis := PsmRef[psmIndex];
            MC_ReadStatus_0[psmIndex+AXIS_NUMBER+MASTER_NUMBER+SLAVE_NUMBER].Enable := TRUE;
        END_FOR

        ErrorStep := STATE_WAIT;
        AcknowledgeStep := STATE_ERROR_SCAN;

        (* End of STATE_CONFIG_FBS *)

(*************************** CHECK_AXES_FOR_ERROR *******************)
    STATE_WAIT: (* check if at least on one of the axes an error occured *)
        IF ((MC_BR_AxisErrorCollector_0.AxisError = TRUE) OR
            (MC_BR_AxisErrorCollector_0.AxisWarning = TRUE) OR
            (MC_BR_AxisErrorCollector_0.FunctionBlockError = TRUE) OR
            (MC_BR_AxisErrorCollector_0.Errorstop = TRUE)) THEN
              ErrorStep := STATE_ERROR_HANDLING;
        ELSE
            GlobalError.AxisTyp := '';
            GlobalError.AxisIndex := 0;
            GlobalError.ErrorRecord.Info := 0;
            GlobalError.ErrorRecord.Number := 0;
            GlobalError.ErrorRecord.ParID := 0;
            GlobalError.ErrorText[0] := '';
            GlobalError.ErrorText[1] := '';
            GlobalError.ErrorText[2] := '';
            GlobalError.ErrorText[3] := '';
        END_IF

        (* End of STATE_WAIT *)

(**************************** HANDLE_ACTIVE_ERRORS ******************)
    STATE_ERROR_HANDLING: (* check witch axis is in ErrorStop and withc axes has to be stopped *)
        (* check if a single axis has to be stopped *)
        FOR axisIndex := 0 TO (AXIS_MAX_INDEX) BY 1 DO
            IF (MC_ReadStatus_0[axisIndex].Errorstop = TRUE) THEN
                Axis[axisIndex].Command.Stop := TRUE;
            END_IF
        END_FOR

        (* check if the master slave combination has to be stopped *)
        FOR masterIndex := 0 TO (MASTER_MAX_INDEX) BY 1 DO
            IF (MC_ReadStatus_0[masterIndex+AXIS_NUMBER].Errorstop = TRUE) THEN
                FOR masterIndex := 0 TO (MASTER_MAX_INDEX) BY 1 DO
                    Master[masterIndex].Command.Stop := TRUE;
                END_FOR

                FOR slaveIndex := 0 TO (SLAVE_MAX_INDEX) BY 1 DO
                    Slave[slaveIndex].Command.Stop := TRUE;
                END_FOR
            END_IF
        END_FOR

        (* check if the master slave combination has to be stopped *)
        FOR slaveIndex := 0 TO (SLAVE_MAX_INDEX) BY 1 DO
            IF  (MC_ReadStatus_0[slaveIndex+AXIS_NUMBER+MASTER_NUMBER].Errorstop = TRUE) THEN
                FOR masterIndex := 0 TO (MASTER_MAX_INDEX) BY 1 DO
                    Master[masterIndex].Command.Stop := TRUE;
                END_FOR

                FOR slaveIndex := 0 TO (SLAVE_MAX_INDEX) BY 1 DO
                    Slave[slaveIndex].Command.Stop := TRUE;
                END_FOR
            END_IF
        END_FOR

    (******************* STEP_SEQUENCE OF ERROR ACKNOWLEDGE *************)
    CASE AcknowledgeStep OF
        (************************** SEARCH FOR ERRORS ***********************)
        STATE_ERROR_SCAN: (* check if an error is active on one of the axis *)
            ErrorStep := STATE_WAIT;
            FOR totalAxisIndex := 0 TO (TOTAL_AXES-1) BY 1 DO
                IF ((MC_BR_ReadAxisError_0[totalAxisIndex].AxisErrorCount > 0) OR
                    (MC_BR_ReadAxisError_0[totalAxisIndex].AxisWarningCount > 0) OR
                    (MC_BR_ReadAxisError_0[totalAxisIndex].FunctionBlockErrorCount > 0)) THEN
                    AcknowledgeStep := STATE_ERROR_ACKNOWLEDGE;
                    ErrorStep := STATE_ERROR_HANDLING;
                    EXIT;
                ELSIF (MC_ReadStatus_0[totalAxisIndex].Errorstop = TRUE) THEN
                    AcknowledgeStep := STATE_RESET;
                    ErrorStep := STATE_ERROR_HANDLING;
                    EXIT;
                END_IF
            END_FOR

            (* End of STATE_ERROR_SCAN *)

        (********************** WAIT FOR ACKNOWLEDGE ************************)
        STATE_ERROR_ACKNOWLEDGE:
            (* copy the actual error information to the global error structure *)
            IF (totalAxisIndex < AXIS_NUMBER) THEN
                GlobalError.AxisTyp := 'Axis';
                GlobalError.ErrorText := Axis[totalAxisIndex].Error.ErrorText;
                GlobalError.ErrorRecord := Axis[totalAxisIndex].Error.ErrorRecord;
            ELSIF (totalAxisIndex < (AXIS_NUMBER+MASTER_NUMBER)) THEN
                GlobalError.AxisTyp := 'Master';
                GlobalError.ErrorText := Master[totalAxisIndex-AXIS_NUMBER].Error.ErrorText;
                GlobalError.ErrorRecord := Master[totalAxisIndex-AXIS_NUMBER].Error.ErrorRecord;
            ELSIF (totalAxisIndex < (AXIS_NUMBER+MASTER_NUMBER+SLAVE_NUMBER)) THEN
                GlobalError.AxisTyp := 'Slave';
                GlobalError.ErrorText := Slave[totalAxisIndex-(AXIS_NUMBER+MASTER_NUMBER)].Error.ErrorText;
                GlobalError.ErrorRecord := Slave[totalAxisIndex-(AXIS_NUMBER+MASTER_NUMBER)].Error.ErrorRecord;
            ELSIF (totalAxisIndex < (AXIS_NUMBER+MASTER_NUMBER+SLAVE_NUMBER+PSM_NUMBER)) THEN
                GlobalError.AxisTyp := 'PSM';
                GlobalError.ErrorText := PowerSupply[totalAxisIndex-(AXIS_NUMBER+MASTER_NUMBER+SLAVE_NUMBER)].Error.ErrorText;
                GlobalError.ErrorRecord := PowerSupply[totalAxisIndex-(AXIS_NUMBER+MASTER_NUMBER+SLAVE_NUMBER)].Error.ErrorRecord;
            END_IF
            GlobalError.AxisIndex := totalAxisIndex;

            IF (GlobalCommand.ErrorAcknowledge = TRUE) THEN
                GlobalCommand.ErrorAcknowledge := FALSE;
                MC_BR_ReadAxisError_0[totalAxisIndex].Acknowledge := TRUE;
            ELSIF (MC_BR_ReadAxisError_0[totalAxisIndex].Acknowledge = TRUE) THEN
                MC_BR_ReadAxisError_0[totalAxisIndex].Acknowledge := FALSE;
                AcknowledgeStep := STATE_ERROR_SCAN;
            END_IF

            (* End of STATE_ERROR_ACKNOWLEDGE *)

        (************************* RESET AXES IN ERRORSTEP ******************)
        STATE_RESET:
            IF (totalAxisIndex < AXIS_NUMBER) THEN
                MC_Reset_0.Axis := AxisRef[totalAxisIndex];
            ELSIF (totalAxisIndex < (AXIS_NUMBER+MASTER_NUMBER)) THEN
                MC_Reset_0.Axis := MasterRef[totalAxisIndex-AXIS_NUMBER];
            ELSIF (totalAxisIndex < (AXIS_NUMBER+MASTER_NUMBER+SLAVE_NUMBER)) THEN
                MC_Reset_0.Axis := SlaveRef[totalAxisIndex-(AXIS_NUMBER+MASTER_NUMBER)];
            ELSE
                MC_Reset_0.Axis := PsmRef[totalAxisIndex-(AXIS_NUMBER+MASTER_NUMBER+SLAVE_NUMBER)];
            END_IF
            MC_Reset_0.Execute := TRUE;

            IF (MC_Reset_0.Done = TRUE) THEN
                MC_Reset_0.Execute := 0;
                AcknowledgeStep := STATE_ERROR_SCAN;
            END_IF

            (* End of STATE_RESET *)
    END_CASE
    (************* END OF STEP SEQUENCE OF ERROR ACKNOWLEDGE ************)

    (* End of STATE_ERROR_HANDLING *)

(****************** DEACTIVATE USED FBS IN CASE OF ERROR ************)
    STATE_INTERNAL_ERROR:
        MC_BR_AxisErrorCollector_0.Enable := FALSE;
        MC_Reset_0.Execute := FALSE;

        FOR configAxisIndex := 0 TO (TOTAL_AXES-1) BY 1 DO
            MC_BR_ReadAxisError_0[configAxisIndex].Enable := FALSE;
            MC_ReadStatus_0[configAxisIndex].Enable := FALSE;
        END_FOR

        ErrorStep := STATE_CONFIG_FBS;

        (* End of STATE_INTERNAL_ERROR *)

END_CASE

(************************** CALL FBS ********************************)
MC_BR_AxisErrorCollector_0();

FOR configAxisIndex := 0 TO TOTAL_AXES BY 1 DO
    MC_BR_ReadAxisError_0[configAxisIndex]();
    IF (configAxisIndex < AXIS_NUMBER) THEN
        Axis[configAxisIndex].Error.AxisErrorCount := MC_BR_ReadAxisError_0[configAxisIndex].AxisErrorCount;
        Axis[configAxisIndex].Error.AxisWarningCount := MC_BR_ReadAxisError_0[configAxisIndex].AxisWarningCount;
        Axis[configAxisIndex].Error.FunctionBlockErrorCount := MC_BR_ReadAxisError_0[configAxisIndex].FunctionBlockErrorCount;
        Axis[configAxisIndex].Error.ErrorRecord := MC_BR_ReadAxisError_0[configAxisIndex].ErrorRecord;
    ELSIF (configAxisIndex < (AXIS_NUMBER+MASTER_NUMBER)) THEN
        Master[configAxisIndex-AXIS_NUMBER].Error.AxisErrorCount := MC_BR_ReadAxisError_0[configAxisIndex].AxisErrorCount;
        Master[configAxisIndex-AXIS_NUMBER].Error.AxisWarningCount := MC_BR_ReadAxisError_0[configAxisIndex].AxisWarningCount;
        Master[configAxisIndex-AXIS_NUMBER].Error.FunctionBlockErrorCount := MC_BR_ReadAxisError_0[configAxisIndex].FunctionBlockErrorCount;
        Master[configAxisIndex-AXIS_NUMBER].Error.ErrorRecord := MC_BR_ReadAxisError_0[configAxisIndex].ErrorRecord;
	ELSIF (configAxisIndex < (AXIS_NUMBER+MASTER_NUMBER+SLAVE_NUMBER)) THEN
		Slave[configAxisIndex-(AXIS_NUMBER+MASTER_NUMBER)].Error.AxisErrorCount := MC_BR_ReadAxisError_0[configAxisIndex].AxisErrorCount;
		Slave[configAxisIndex-(AXIS_NUMBER+MASTER_NUMBER)].Error.AxisWarningCount := MC_BR_ReadAxisError_0[configAxisIndex].AxisWarningCount;
		Slave[configAxisIndex-(AXIS_NUMBER+MASTER_NUMBER)].Error.FunctionBlockErrorCount := MC_BR_ReadAxisError_0[configAxisIndex].FunctionBlockErrorCount;
		Slave[configAxisIndex-(AXIS_NUMBER+MASTER_NUMBER)].Error.ErrorRecord := MC_BR_ReadAxisError_0[configAxisIndex].ErrorRecord;
	ELSIF (configAxisIndex < (AXIS_NUMBER+MASTER_NUMBER+SLAVE_NUMBER+PSM_NUMBER)) THEN
		PowerSupply[configAxisIndex-(AXIS_NUMBER+MASTER_NUMBER+SLAVE_NUMBER)].Error.AxisErrorCount := MC_BR_ReadAxisError_0[configAxisIndex].AxisErrorCount;
        PowerSupply[configAxisIndex-(AXIS_NUMBER+MASTER_NUMBER+SLAVE_NUMBER)].Error.AxisWarningCount := MC_BR_ReadAxisError_0[configAxisIndex].AxisWarningCount;
        PowerSupply[configAxisIndex-(AXIS_NUMBER+MASTER_NUMBER+SLAVE_NUMBER)].Error.FunctionBlockErrorCount := MC_BR_ReadAxisError_0[configAxisIndex].FunctionBlockErrorCount;
        PowerSupply[configAxisIndex-(AXIS_NUMBER+MASTER_NUMBER+SLAVE_NUMBER)].Error.ErrorRecord := MC_BR_ReadAxisError_0[configAxisIndex].ErrorRecord;
    END_IF
    MC_ReadStatus_0[configAxisIndex]();
END_FOR

MC_Reset_0();

END_PROGRAM
```

#### errorHandlingInit.st - Initialization code
```iecst
(********************************************************************
 * COPYRIGHT -- Bernecker + Rainer
 ********************************************************************
 * Program: ErrorHandling
 * File: errorHandlingInit.st
 * Author: Bernecker + Rainer
 * Created: March 01, 2011
 ********************************************************************
  * Implementation OF PROGRAM ErrorHandling
 ********************************************************************)

PROGRAM _INIT
    AcknowledgeStep := STATE_ERROR_SCAN;
END_PROGRAM
```

#### errorHandling.var - Local variables
```iecst
(*Index variables*)
VAR
	configAxisIndex : USINT; (*count variable for configurating "for"-loops*)
	totalAxisIndex : USINT; (*count variable for all axes acting "for"-loops*)
	psmIndex : USINT;
	axisIndex : USINT; (*count variable for single axes acting "for"-loops*)
	masterIndex : USINT; (*count variable for master axes acting "for"-loops*)
	slaveIndex : USINT; (*count variable for slave axes acting "for"-loops*)
END_VAR
(*Actual steps inside the step sequences*)
VAR
	ErrorStep : USINT; (*current step in the step sequence*)
	AcknowledgeStep : USINT; (*current step in the acknowledge step sequence *)
END_VAR
(*Error Steps*)
VAR CONSTANT
	STATE_CONFIG_FBS : USINT := 0; (*constant for the step in which the function blocks are configured*)
	STATE_WAIT : USINT := 1; (*constant for the step in which it is waited for a occuring error*)
	STATE_ERROR_HANDLING : USINT := 2; (*constant for the step in which all necessary axes are stopped *)
	STATE_INTERNAL_ERROR : USINT := 3; (*constant for the step in which all function blocks are disabled in case of an FB error*)
END_VAR
(*Acknowledge Steps*)
VAR CONSTANT
	STATE_ERROR_SCAN : USINT := 10; (*constant for the step in which the first active is searched*)
	STATE_ERROR_ACKNOWLEDGE : USINT := 11; (*constant for the step in which the actual output error is acknowledged after user command*)
	STATE_RESET : USINT := 12; (*constant for the step in which the axes are reset after all errors where acknowled*)
END_VAR
(*Function Blocks*)
VAR
	MC_BR_AxisErrorCollector_0 : MC_BR_AxisErrorCollector; (*Function Block*)
	MC_BR_ReadAxisError_0 : ARRAY[0..TOTAL_AXES] OF MC_BR_ReadAxisError; (*Function Block*)
	MC_ReadStatus_0 : ARRAY[0..TOTAL_AXES] OF MC_ReadStatus; (*Function Block*)
	MC_Reset_0 : MC_Reset; (*Function Block*)
END_VAR
```

### Program Logical/MotionControl/AxisControl/VMaster (IEC)

- Cyclic.st (reference to Logical/Template/Axis/GenericVirtualAxis/Cyclic.st)

- Act_Config.st (reference to Logical/Template/Axis/GenericVirtualAxis/Act_Config.st)

#### Act_Parameters.st
```iecst
ACTION Act_Parameters:

	//---- Numero del Eje ----///
	AxisIndex 		:= VMASTER;

	//---- MpLink ----//
	MpLink 			:= gVMasterLink;
	Axis 			:= ADR(gVMaster);
	//MpLinkMaster;

	//---- Nombre del eje ----//
	AxisName 		:= 'Eje Generico';

	//---- Hablita el eje ----//
	gAxis[AxisIndex].Command.Enable := TRUE; // ESTE DATA DEBERA SER USADO EN UN VARIABLE DE LA CONFIGURACION MAQUINA PARA HABILITAR O DESHABILITAR UN EJE.

	//---- Limite de velocidad -----//
	LimitSpeed 		:= 6600.0;

	//----- Limete de aceleracion/desaceleracion ----//
	LimitAccDec 	:= 6600.0;

	//---- Relacion de velocoidad motor/reductor ----//
	GearIn 			:= 1;
	GearOut 		:= 1;

	//---- Seleccion direccion de rotacion del eje ----//
	AxisDirection := TRUE; // TRUE = sentido de las manesillas del reloj; FALSE = en contra de las manesillas del reloj;

	// ---- Definicion Paramentros de posicion del eje ----//
	HeadNumber 		:= 1;
	Period 			:= 360.0 * HeadNumber;
	SectorNumber 	:= 1;
	Resolution		:= 0.01;

END_ACTION
```

- Variables.var (reference to Logical/Template/Axis/GenericVirtualAxis/Variables.var)

#### Act_Config.st - not listed in the package file held
```iecst
ACTION Act_Config:

	//---- Numero del Eje ----///
	AxisIndex := VMASTER;

	//---- MpLink ----//
	MpLink 			:= gVMasterLink;
	Axis 			:= ADR(gVMaster);
	//MpLinkMaster;

	//---- Nombre del eje ----//
	AxisName := 'Eje Generico';

	//---- Hablita el eje ----//
	gAxis[AxisIndex].Command.Enable := TRUE; // ESTE DATA DEBERA SER USADO EN UN VARIABLE DE LA CONFIGURACION MAQUINA PARA HABILITAR O DESHABILITAR UN EJE.

	//---- Limite de velocidad -----//
	LimitSpeed 	:= 6600.0;

	//----- Limete de aceleracion/desaceleracion ----//
	LimitAccDec := 6600.0;

	//---- Relacion de velocoidad motor/reductor ----//
	GearIn 	:= 1;
	GearOut := 1;

	//---- Seleccion direccion de rotacion del eje ----//
	AxisDirection := TRUE; // TRUE = sentido de las manesillas del reloj; FALSE = en contra de las manesillas del reloj;

	// ---- Definicion sentido de giro del eje ----//
	IF AxisDirection THEN
		Direction	:= mpAXIS_DIR_CLOCKWISE;
	ELSE
		Direction	:= mpAXIS_DIR_COUNTERCLOCKWISE;
	END_IF

	// ---- Definicion Paramentros de posicion del eje ----//
	HeadNumber 			:= 1;
	Period 				:= 360.0 * HeadNumber;
	SectorNumber 		:= 1;
	Resolution			:= 0.01;
	/////////////////////////////////////////////////////////////////

	(**** Secuencia configuarcion Eje *****)

	IF NOT ConfigReq THEN
		StConfig := CONFIG_WAIT;
	END_IF

	CASE StConfig OF

		CONFIG_WAIT:

			IF ConfigReq THEN
				StConfig := CONFIG_LOAD_REQ;
			END_IF

		CONFIG_LOAD_REQ:

			(* Carga la configuracion por default en Confing.mpaxisbasic*)

			AxisConfig.Load	:= TRUE;

			IF AxisConfig.CommandDone THEN
				StConfig := CONFIG_LOAD_DONE;
			END_IF

		CONFIG_LOAD_DONE:

			(* Actualiza la configuracion, carga parametros asignados por el usuario *)

			AxisConfig.Load	:= FALSE;
			StConfig := CONFIG_SAVE_REQ;

		CONFIG_SAVE_REQ:

			AxisConfigPar.AxisName := AxisName ;

			//Axis
			AxisConfigPar.Axis.BaseType 				:= mpAXIS_PERIODIC_ROTARY;
			AxisConfigPar.Axis.MeasurementUnit 			:= mpAXIS_UNIT_GENERIC;
			AxisConfigPar.Axis.MeasurementResolution 	:= Resolution;
			AxisConfigPar.Axis.PeriodSettings.Period	:= Period;

			AxisConfigPar.Axis.MovementLimits.VelocityPositive	:= LimitSpeed;
			AxisConfigPar.Axis.MovementLimits.VelocityNegative	:= LimitSpeed;
			AxisConfigPar.Axis.MovementLimits.Acceleration		:= LimitAccDec;
			AxisConfigPar.Axis.MovementLimits.Deceleration		:= LimitAccDec;

			//Drive
			AxisConfigPar.Drive.Gearbox.Input			:= GearIn;
			AxisConfigPar.Drive.Gearbox.Output			:= GearOut;
			AxisConfigPar.Drive.Gearbox.Direction 		:= Direction;
			AxisConfigPar.Drive.Transformation.ReferenceDistance := Period * SectorNumber;

			(* Salva en el drive los parametros asignados por el usuario *)

			AxisConfig.Save := TRUE;

			IF AxisConfig.CommandDone THEN
				StConfig := CONFIG_SAVE_DONE;
			END_IF

		CONFIG_SAVE_DONE:

			(* Configuracion terminada *)

			AxisConfig.Save := FALSE;
			ConfigReq		:= FALSE;
			ConfigDone		:= TRUE;

	END_CASE

	//	gAxis[AxisIndex].Cmd.ConfigReq := StConfig = CONFIG_LOAD_REQ;
	//	gAxis[AxisIndex].Sts.ConfigDone := StConfig = CONFIG_SAVE_DONE;

	AxisBasic.Enable 	:= gAxis[AxisIndex].Command.Enable;
	AxisConfig.Enable 	:= AxisBasic.Active;

	(********** FB's Configuration *********)

	AxisBasic.Axis 		:= Axis;
	AxisBasic.MpLink 	:= ADR(MpLink);
	AxisBasic.Parameters := ADR(AxisBasicPar);

	AxisConfig.MpLink 			:= ADR(MpLink);
	AxisConfig.Configuration 	:= ADR(AxisConfigPar);

	//	AxisCam.MpLink				:= ADR(MpLink);
	//	AxisCam.MpLinkMaster		:= ADR(MpLinkMaster);
	//	AxisCam.Parameters			:= ADR(AxisCamPar);

	(****************************************)

END_ACTION
```

### Program Logical/MotionControl/AxisControl/Reel_A (IEC)

- Cyclic.st (reference to Logical/Template/Axis/GenericAxis/Cyclic.st)

- Act_Config.st (reference to Logical/Template/Axis/GenericAxis/Act_Config.st)

#### Act_Parameters.st
```iecst
ACTION Act_Parameters:

	//---- Numero del Eje ----///
	AxisIndex := REEL_A;

	//---- MpLink ----//

	Axis 			:= ADR(gAxReel_A);
	MpLinkMaster    := gVMasterLink;
	MpLink 			:= gAxReelA_Link;

	//---- Nombre del eje ----//
	AxisName := 'Reel A';

	//---- Hablita el eje ----//
	gAxis[AxisIndex].Command.Enable := TRUE; // ESTE DATA DEBERA SER USADO EN UN VARIABLE DE LA CONFIGURACION MAQUINA PARA HABILITAR O DESHABILITAR UN EJE.

	//---- Limite de velocidad -----//
	LimitSpeed 	:= 6600.0;

	//----- Limete de aceleracion/desaceleracion ----//
	LimitAccDec := 6600.0;

	//---- Relacion de velocoidad motor/reductor ----//
	GearIn 	:= 1;
	GearOut := 1;

	//---- Seleccion direccion de rotacion del eje ----//
	AxisDirection := TRUE; // TRUE = sentido de las manesillas del reloj; FALSE = en contra de las manesillas del reloj;

	// ---- Definicion Paramentros de posicion del eje ----//
	HeadNumber 			:= 1;
	Period 				:= 360.0 * HeadNumber;
	SectorNumber 		:= 1;
	Resolution			:= 0.01;
	/////////////////////////////////////////////////////////////////

END_ACTION
```

- Types.typ (reference to Logical/Template/Axis/GenericAxis/Types.typ)

- Variables.var (reference to Logical/Template/Axis/GenericAxis/Variables.var)

#### Act_Config.st - not listed in the package file held
```iecst
ACTION Act_Config:

	//---- Numero del Eje ----///
	AxisIndex := REEL_A;

	//---- MpLink ----//
	MpLink 			:= gAxReelA_Link;
	Axis 			:= ADR(gAxReel_A);
	//MpLinkMaster;

	//---- Nombre del eje ----//
	AxisName := 'Reel A';

	//---- Hablita el eje ----//
	gAxis[AxisIndex].Command.Enable := TRUE; // ESTE DATA DEBERA SER USADO EN UN VARIABLE DE LA CONFIGURACION MAQUINA PARA HABILITAR O DESHABILITAR UN EJE.

	//---- Limite de velocidad -----//
	LimitSpeed 	:= 6600.0;

	//----- Limete de aceleracion/desaceleracion ----//
	LimitAccDec := 6600.0;

	//---- Relacion de velocoidad motor/reductor ----//
	GearIn 	:= 1;
	GearOut := 1;

	//---- Seleccion direccion de rotacion del eje ----//
	AxisDirection := TRUE; // TRUE = sentido de las manesillas del reloj; FALSE = en contra de las manesillas del reloj;

	// ---- Definicion sentido de giro del eje ----//
	IF AxisDirection THEN
		Direction	:= mpAXIS_DIR_CLOCKWISE;
	ELSE
		Direction	:= mpAXIS_DIR_COUNTERCLOCKWISE;
	END_IF

	// ---- Definicion Paramentros de posicion del eje ----//
	HeadNumber 			:= 1;
	Period 				:= 360.0 * HeadNumber;
	SectorNumber 		:= 1;
	Resolution			:= 0.01;
	/////////////////////////////////////////////////////////////////

	(**** Secuencia configuarcion Eje *****)

	IF NOT ConfigReq THEN
		StConfig := CONFIG_WAIT;
	END_IF

	CASE StConfig OF

		CONFIG_WAIT:

			IF ConfigReq THEN
				StConfig := CONFIG_LOAD_REQ;
			END_IF

		CONFIG_LOAD_REQ:

			(* Carga la configuracion por default en Confing.mpaxisbasic*)

			AxisConfig.Load	:= TRUE;

			IF AxisConfig.CommandDone THEN
				StConfig := CONFIG_LOAD_DONE;
			END_IF

		CONFIG_LOAD_DONE:

			(* Actualiza la configuracion, carga parametros asignados por el usuario *)

			AxisConfig.Load	:= FALSE;
			StConfig := CONFIG_SAVE_REQ;

		CONFIG_SAVE_REQ:

			AxisConfigPar.AxisName := AxisName ;

			//Axis
			AxisConfigPar.Axis.BaseType 				:= mpAXIS_PERIODIC_ROTARY;
			AxisConfigPar.Axis.MeasurementUnit 			:= mpAXIS_UNIT_GENERIC;
			AxisConfigPar.Axis.MeasurementResolution 	:= Resolution;
			AxisConfigPar.Axis.PeriodSettings.Period	:= Period;

			AxisConfigPar.Axis.MovementLimits.VelocityPositive	:= LimitSpeed;
			AxisConfigPar.Axis.MovementLimits.VelocityNegative	:= LimitSpeed;
			AxisConfigPar.Axis.MovementLimits.Acceleration		:= LimitAccDec;
			AxisConfigPar.Axis.MovementLimits.Deceleration		:= LimitAccDec;

			//Drive
			AxisConfigPar.Drive.Gearbox.Input			:= GearIn;
			AxisConfigPar.Drive.Gearbox.Output			:= GearOut;
			AxisConfigPar.Drive.Gearbox.Direction 		:= Direction;
			AxisConfigPar.Drive.Transformation.ReferenceDistance := Period * SectorNumber;

			(* Salva en el drive los parametros asignados por el usuario *)

			AxisConfig.Save := TRUE;

			IF AxisConfig.CommandDone THEN
				StConfig := CONFIG_SAVE_DONE;
			END_IF

		CONFIG_SAVE_DONE:

			(* Configuracion terminada *)

			AxisConfig.Save := FALSE;
			ConfigReq		:= FALSE;
			ConfigDone		:= TRUE;

	END_CASE

	//	gAxis[AxisIndex].Cmd.ConfigReq := StConfig = CONFIG_LOAD_REQ;
	//	gAxis[AxisIndex].Sts.ConfigDone := StConfig = CONFIG_SAVE_DONE;

	AxisBasic.Enable 	:= gAxis[AxisIndex].Command.Enable;
	AxisConfig.Enable 	:= AxisBasic.Active;

	(********** FB's Configuration *********)

	AxisBasic.Axis 		:= Axis;
	AxisBasic.MpLink 	:= ADR(MpLink);
	AxisBasic.Parameters := ADR(AxisBasicPar);

	AxisConfig.MpLink 			:= ADR(MpLink);
	AxisConfig.Configuration 	:= ADR(AxisConfigPar);

	//	AxisCam.MpLink				:= ADR(MpLink);
	//	AxisCam.MpLinkMaster		:= ADR(MpLinkMaster);
	//	AxisCam.Parameters			:= ADR(AxisCamPar);

	(****************************************)

END_ACTION
```

### Program Logical/MotionControl/AxisControl/Reel_B (IEC)

- Cyclic.st (reference to Logical/Template/Axis/GenericAxis/Cyclic.st)

- Act_Config.st (reference to Logical/Template/Axis/GenericAxis/Act_Config.st)

#### Act_Parameters.st
```iecst
ACTION Act_Parameters:

//---- Numero del Eje ----///
	AxisIndex := REEL_B;

	//---- MpLink ----//

	Axis 			:= ADR(gAxReel_B);
	MpLinkMaster    := gVMasterLink;
	MpLink 			:= gAxReelB_Link;

	//---- Nombre del eje ----//
	AxisName := 'Reel B';

	//---- Hablita el eje ----//
	gAxis[AxisIndex].Command.Enable := TRUE; // ESTE DATA DEBERA SER USADO EN UN VARIABLE DE LA CONFIGURACION MAQUINA PARA HABILITAR O DESHABILITAR UN EJE.

	//---- Limite de velocidad -----//
	LimitSpeed 	:= 6600.0;

	//----- Limete de aceleracion/desaceleracion ----//
	LimitAccDec := 6600.0;

	//---- Relacion de velocoidad motor/reductor ----//
	GearIn 	:= 1;
	GearOut := 1;

	//---- Seleccion direccion de rotacion del eje ----//
	AxisDirection := TRUE; // TRUE = sentido de las manesillas del reloj; FALSE = en contra de las manesillas del reloj;

	// ---- Definicion Paramentros de posicion del eje ----//
	HeadNumber 			:= 1;
	Period 				:= 360.0 * HeadNumber;
	SectorNumber 		:= 1;
	Resolution			:= 0.01;

END_ACTION
```

- Variables.var (reference to Logical/Template/Axis/GenericAxis/Variables.var)

- Types.typ (reference to Logical/Template/Axis/GenericAxis/Types.typ)

#### Act_Config.st - not listed in the package file held
```iecst
ACTION Act_Config:

	//---- Numero del Eje ----///
	AxisIndex := REEL_B;

	//---- MpLink ----//
	MpLink 			:= gAxReelB_Link;
	Axis 			:= ADR(gAxReel_B);
	//MpLinkMaster;

	//---- Nombre del eje ----//
	AxisName := 'Reel B';

	//---- Hablita el eje ----//
	gAxis[AxisIndex].Command.Enable := TRUE; // ESTE DATA DEBERA SER USADO EN UN VARIABLE DE LA CONFIGURACION MAQUINA PARA HABILITAR O DESHABILITAR UN EJE.

	//---- Limite de velocidad -----//
	LimitSpeed 	:= 6600.0;

	//----- Limete de aceleracion/desaceleracion ----//
	LimitAccDec := 6600.0;

	//---- Relacion de velocoidad motor/reductor ----//
	GearIn 	:= 1;
	GearOut := 1;

	//---- Seleccion direccion de rotacion del eje ----//
	AxisDirection := TRUE; // TRUE = sentido de las manesillas del reloj; FALSE = en contra de las manesillas del reloj;

	// ---- Definicion sentido de giro del eje ----//
	IF AxisDirection THEN
		Direction	:= mpAXIS_DIR_CLOCKWISE;
	ELSE
		Direction	:= mpAXIS_DIR_COUNTERCLOCKWISE;
	END_IF

	// ---- Definicion Paramentros de posicion del eje ----//
	HeadNumber 			:= 1;
	Period 				:= 360.0 * HeadNumber;
	SectorNumber 		:= 1;
	Resolution			:= 0.01;
	/////////////////////////////////////////////////////////////////

	(**** Secuencia configuarcion Eje *****)

	IF NOT ConfigReq THEN
		StConfig := CONFIG_WAIT;
	END_IF

	CASE StConfig OF

		CONFIG_WAIT:

			IF ConfigReq THEN
				StConfig := CONFIG_LOAD_REQ;
			END_IF

		CONFIG_LOAD_REQ:

			(* Carga la configuracion por default en Confing.mpaxisbasic*)

			AxisConfig.Load	:= TRUE;

			IF AxisConfig.CommandDone THEN
				StConfig := CONFIG_LOAD_DONE;
			END_IF

		CONFIG_LOAD_DONE:

			(* Actualiza la configuracion, carga parametros asignados por el usuario *)

			AxisConfig.Load	:= FALSE;
			StConfig := CONFIG_SAVE_REQ;

		CONFIG_SAVE_REQ:

			AxisConfigPar.AxisName := AxisName ;

			//Axis
			AxisConfigPar.Axis.BaseType 				:= mpAXIS_PERIODIC_ROTARY;
			AxisConfigPar.Axis.MeasurementUnit 			:= mpAXIS_UNIT_GENERIC;
			AxisConfigPar.Axis.MeasurementResolution 	:= Resolution;
			AxisConfigPar.Axis.PeriodSettings.Period	:= Period;

			AxisConfigPar.Axis.MovementLimits.VelocityPositive	:= LimitSpeed;
			AxisConfigPar.Axis.MovementLimits.VelocityNegative	:= LimitSpeed;
			AxisConfigPar.Axis.MovementLimits.Acceleration		:= LimitAccDec;
			AxisConfigPar.Axis.MovementLimits.Deceleration		:= LimitAccDec;

			//Drive
			AxisConfigPar.Drive.Gearbox.Input			:= GearIn;
			AxisConfigPar.Drive.Gearbox.Output			:= GearOut;
			AxisConfigPar.Drive.Gearbox.Direction 		:= Direction;
			AxisConfigPar.Drive.Transformation.ReferenceDistance := Period * SectorNumber;

			(* Salva en el drive los parametros asignados por el usuario *)

			AxisConfig.Save := TRUE;

			IF AxisConfig.CommandDone THEN
				StConfig := CONFIG_SAVE_DONE;
			END_IF

		CONFIG_SAVE_DONE:

			(* Configuracion terminada *)

			AxisConfig.Save := FALSE;
			ConfigReq		:= FALSE;
			ConfigDone		:= TRUE;

	END_CASE

	//	gAxis[AxisIndex].Cmd.ConfigReq := StConfig = CONFIG_LOAD_REQ;
	//	gAxis[AxisIndex].Sts.ConfigDone := StConfig = CONFIG_SAVE_DONE;

	AxisBasic.Enable 	:= gAxis[AxisIndex].Command.Enable;
	AxisConfig.Enable 	:= AxisBasic.Active;

	(********** FB's Configuration *********)

	AxisBasic.Axis 		:= Axis;
	AxisBasic.MpLink 	:= ADR(MpLink);
	AxisBasic.Parameters := ADR(AxisBasicPar);

	AxisConfig.MpLink 			:= ADR(MpLink);
	AxisConfig.Configuration 	:= ADR(AxisConfigPar);

	//	AxisCam.MpLink				:= ADR(MpLink);
	//	AxisCam.MpLinkMaster		:= ADR(MpLinkMaster);
	//	AxisCam.Parameters			:= ADR(AxisCamPar);

	(****************************************)

END_ACTION
```

### Program Logical/MotionControl/Winder/LineControl/MainControl (IEC)

#### Types.typ
```iecst
TYPE
	AxisState_enum :
		(
		STATE_WAIT := 0,
		STATE_POWER_ON := 10,
		STATE_ERROR := 20,
		STATE_STOP := 30,
		STATE_READY := 40,
		STATE_HOME := 50,
		STATE_AUTO := 60,
		STATE_MANUAL := 70,
		STATE_MAINT := 80
		);
END_TYPE
```

#### Variables.var
```iecst
VAR
	StLineCtrl : AxisState_enum;
	i : INT;
	Auto : BOOL;
END_VAR
```

#### Main.st
```iecst
PROGRAM _INIT
	(* Insert code here *)

END_PROGRAM

PROGRAM _CYCLIC

	(**** Line control Sequence ****)

	CASE StLineCtrl OF

		STATE_WAIT:

			FOR i:= 0 TO MAX_AXIS DO

				IF gAxis[i].Status.Active THEN
					StLineCtrl:= STATE_POWER_ON;
				END_IF
			END_FOR

		STATE_POWER_ON:

			FOR i := 0 TO MAX_AXIS DO

				gAxis[i].Command.PowerOn := TRUE;

				IF gAxis[i].Status.PoweredOn THEN
					StLineCtrl:= STATE_HOME;
				END_IF

			END_FOR

		STATE_HOME:

			FOR i := 0 TO MAX_AXIS DO

				IF gAxis[i].Status.Homed THEN
					StLineCtrl:= STATE_READY;
				END_IF

			END_FOR

		STATE_READY:

			IF Auto THEN
				StLineCtrl := STATE_AUTO;
			END_IF

		STATE_AUTO:

			FOR i := 0 TO MAX_AXIS DO

				gAxis[i].Command.Auto := TRUE;

				IF NOT Auto THEN
					gAxis[i].Command.Auto := FALSE;
					StLineCtrl	:= STATE_READY;
				END_IF

			END_FOR

	END_CASE

END_PROGRAM

PROGRAM _EXIT
	(* Insert code here *)

END_PROGRAM
```

- Data object Logical/AxisObject/VirtualAxis/VAxInit (Vax) (no source held here)

- Data object Logical/AxisObject/RealAxis/AxInit (Ax) (no source held here)

Listed in the project but not available here: Logical/Template/Axis/GenericAxis/Init.st, Logical/Template/Axis/GenericAxis/Exit.st, Logical/Template/Axis/GenericVirtualAxis/Init.st, Logical/Template/Axis/GenericVirtualAxis/Types.typ, Logical/Template/Axis/GenericAxis/Init.st, Logical/Template/Axis/GenericAxis/Init.st, Logical/AxisObject/acp10etxen, Logical/AxisObject/RealAxis/AcpParTab
